FUNCTION_BLOCK FB_AnalogOut EXTENDS FB_AnalogOutput
VAR_INPUT
END_VAR
VAR_OUTPUT
END_VAR
VAR
END_VAR

END_FUNCTION_BLOCK

(* stored: Version 1.1.0.1, ProductVersion 3.1.4022.18
   POU FB_AnalogOut: Id {53b4ccd0-b970-46d7-b218-47ae86916403}, SpecialFunc None *)
